{attribute 'GeneratedUsingTerminal: EL6090-0000-0016'}
{attribute addProperty BoxType "EL6090-0000-0016"}
{attribute addProperty Id "DIS_InputsAT %I*DIS_Inputs_E0E384E36DIS_OutputsAT %Q*DIS_Outputs_6C9BFFEE4WcStateAT %I*WcState_9091E0EB2InfoDataAT %I*InfoData_94A18F5E2"}
{attribute addProperty CRC "2613166276"}
{attribute addProperty Size "14"}
TYPE EL6090_9BC1C0C4 EXTENDS EtcSlaveTerminalBase_947E5A46 :
STRUCT
	{attribute addProperty Name "DIS_Inputs"}
	DIS_Inputs : DIS_Inputs_E0E384E3;
	{attribute addProperty Name "DIS_Outputs"}
	DIS_Outputs : DIS_Outputs_6C9BFFEE;
	{attribute addProperty Name "WcState"}
	WcState : WcState_9091E0EB;
	{attribute addProperty Name "InfoData"}
	InfoData : InfoData_94A18F5E;
END_STRUCT
END_TYPE

(* stored: Version 1.2.0.0, ProductVersion 3.1.4024.9
   DUT EL6090_9BC1C0C4: Id {59be29d0-9053-46fb-98cc-6339c0c4265f} *)
